{attribute addProperty BoxType "EK1122-0000-0018"}
{attribute addProperty Id "Beckhoff_EL9xxxsub_EK1100EK1100_179A0949162"}
{attribute addProperty CRC "759803653"}
{attribute addProperty SizeInBites "16"}
{attribute addProperty SizeInBytes "2"}
TYPE Beckhoff_EL9xxxEK1122_2D49AF05 EXTENDS EK1122_179A0949 :
STRUCT
	{attribute addProperty Name "Beckhoff_EL9xxxsub_EK1100"}
	Beckhoff_EL9xxxsub_EK1100 : EK1100_179A0949;
END_STRUCT
END_TYPE

(* stored: Version 1.2.0.0, ProductVersion 3.1.4024.9
   DUT Beckhoff_EL9xxxEK1122_2D49AF05: Id {7b7d8069-a2ed-47dc-934a-5395e40d9e1d} *)
